FUNCTION_BLOCK "FB_ProductTrigger"
{ S7_Optimized_Access := 'FALSE' }
VERSION : 0.1
   VAR_INPUT
      SensorInput : Bool;
      TimeDelay : Time;
      SystemTime : Time;
   END_VAR

   VAR_OUTPUT
      TriggerMovement : Bool;
      ProductCount : Int;
   END_VAR

   VAR_TEMP
      ProductQueue : Array[0..1] of "ProductEntry";
      SensorMemory : Bool;
      i : Int;
   END_VAR


BEGIN
	// Reset output
	#TriggerMovement := FALSE;

	// Flankdetectie op sensor
	IF #SensorInput AND NOT #SensorMemory THEN
	    // Zoek eerste vrije plek
	    FOR #i := 1 TO 10 DO
	        IF NOT #ProductQueue[#i].Active THEN
	            #ProductQueue[#i].Active := TRUE;
	            #ProductQueue[#i].StartTime := #SystemTime;
	            EXIT;
	        END_IF;
	    END_FOR;
	END_IF;
	#SensorMemory := #SensorInput;

	// Kijk of een van de producten klaar is voor beweging
	FOR #i := 1 TO 10 DO
	    IF #ProductQueue[#i].Active AND (#SystemTime - #ProductQueue[#i].StartTime >= #TimeDelay) THEN
	        #TriggerMovement := TRUE;
	        #ProductQueue[#i].Active := FALSE; // Verwijder uit wachtrij
	        EXIT; // Eén tegelijk
	    END_IF;
	END_FOR;

	// Update productenteller
	#ProductCount := 0;
	FOR #i := 1 TO 10 DO
	    IF #ProductQueue[#i].Active THEN
	        #ProductCount := #ProductCount + 1;
	    END_IF;
	END_FOR;

END_FUNCTION_BLOCK

